// TIA Portal project "FactoryIO_Template_S7-1200_V16_V16" (V16)
// Vorlageprojekt für das Buch mit Zielsystem S7-1200

(* hardware
DEVICE "S7-1200-Station_1"  S7-1200 Station
   slot 0: "Baugruppenträger_0"  Rack  V1.0
   slot 1: "PLC_1"  CPU 1211C DC/DC/DC  6ES7 211-1AE40-0XB0  V4.1
*)

// ===== PLC "PLC_1"  CPU 1211C DC/DC/DC =====

VAR_GLOBAL   // PLC tag table "Standard-Variablentabelle"
   "6m" AT %A0.0 : Bool;
   "start" AT %E0.0 : Bool;
   "stop" AT %E0.1 : Bool;
   "Tag_4" AT %I10.0 : Bool;
   "Tag_5" AT %Q10.0 : Bool;
   "Tag_6" AT %I10.1 : Bool;
   "2m 1" AT %Q0.1 : Bool;
   "2m 2" AT %Q0.2 : Bool;
   "2m 3" AT %Q0.3 : Bool;
   "2m 4" AT %Q0.4 : Bool;
   "ccw" AT %Q0.5 : Bool;
   "sensor 4" AT %I0.3 : Bool;
   "sensor 1" AT %I0.2 : Bool;
   "pivot 1" AT %Q0.6 : Bool;
   "pivot 1 +" AT %Q0.7 : Bool;
   "sensor 2" AT %I0.4 : Bool;
   "sensor 3" AT %I0.5 : Bool;
   "pivot 2" AT %Q1.0 : Bool;
   "pivot 2 +" AT %Q1.1 : Bool;
   "pivot 3" AT %Q1.2 : Bool;
   "pivot 3 +" AT %Q1.3 : Bool;
END_VAR

// folder: System blocks/Program resources

DATA_BLOCK "IEC_Timer_0_DB"   // DB1
{ S7_Optimized_Access := 'TRUE' }
AUTHOR : Simatic
FAMILY : IEC
NAME : IEC_TMR
VERSION : 1.0
// stored: InstanceOfName IEC_TIMER
"IEC_TIMER"
BEGIN
END_DATA_BLOCK

DATA_BLOCK "IEC_Timer_0_DB_1"   // DB2
{ S7_Optimized_Access := 'TRUE' }
AUTHOR : Simatic
FAMILY : IEC
NAME : IEC_TMR
VERSION : 1.0
// stored: InstanceOfName IEC_TIMER
"IEC_TIMER"
BEGIN
END_DATA_BLOCK

DATA_BLOCK "IEC_Timer_0_DB_2"   // DB3
{ S7_Optimized_Access := 'TRUE' }
AUTHOR : Simatic
FAMILY : IEC
NAME : IEC_TMR
VERSION : 1.0
// stored: InstanceOfName IEC_TIMER
"IEC_TIMER"
BEGIN
END_DATA_BLOCK

// folder: (top level)

FUNCTION "MHJ-PLC-Lab-Function-S71200" : Void   // FC9000, SCL
{ S7_Optimized_Access := 'TRUE' }
VERSION : 0.1
   VAR_TEMP
      rdTimeReturn : Int;
      outputTime : DTL;
      SyncVal : Byte;
      forVal : Int;
      forVal_2 : Int;
      Value : Byte;
   END_VAR
   VAR CONSTANT
      CompVal : Byte := 16#34;
      Value_01 : Byte := 16#11;
      Value_01_DW : DWord := 16#A165_D992;
      Value_02_DW : DWord := 16#58BE_4401;
   END_VAR
BEGIN

   #Value:=PEEK(area := 16#82,
        dbNumber := 0,
        byteOffset := 511);
   #Value := #Value + 1;

   POKE(area := 16#82,
        dbNumber := 0,
        byteOffset := 511,
        value := #Value);

   POKE(area:=16#81,
        dbNumber:=0,
        byteOffset:=1016,
        value:=#Value_01_DW);
   POKE(area := 16#81,
        dbNumber := 0,
        byteOffset := 1020,
        value := #Value_02_DW);

   POKE(area := 16#81,
        dbNumber := 0,
        byteOffset := 511,
        value := B#16#00);

   FOR #forVal := 0 TO 120 DO
       FOR #forVal_2:=0 TO 10 DO
           #rdTimeReturn:=RD_SYS_T(#outputTime);
           #rdTimeReturn := WR_SYS_T(#outputTime);
           #rdTimeReturn := RD_SYS_T(#outputTime);
           #rdTimeReturn := WR_SYS_T(#outputTime);
       END_FOR;
       #SyncVal:= PEEK(area := 16#81,
                      dbNumber := 0,
                      byteOffset := 511);
       IF #SyncVal = #CompVal THEN
          GOTO M_1;
       END_IF;
   END_FOR;
   RETURN;

   M_1:
   POKE(area := 16#81,
        dbNumber := 0,
        byteOffset := 511,
        value := B#16#0);
END_FUNCTION

ORGANIZATION_BLOCK "Main"   // OB1, LAD, ProgramCycle
TITLE = "Main Program Sweep (Cycle)"
{ S7_Optimized_Access := 'TRUE' }
VERSION : 0.1
   VAR_INPUT
      Initial_Call : Bool;   // Initial call of this OB
      Remanence : Bool;   // =True, if remanent data are available
   END_VAR
BEGIN

REGION Network 1: Konnektierungsbaustein für PLC-Lab
   // Im Netzwerk 1 wird der Konnektierungsbaustein für PLC-Lab aufgerufen.
   // Dieser Aufruf darf nicht entfernt werden!
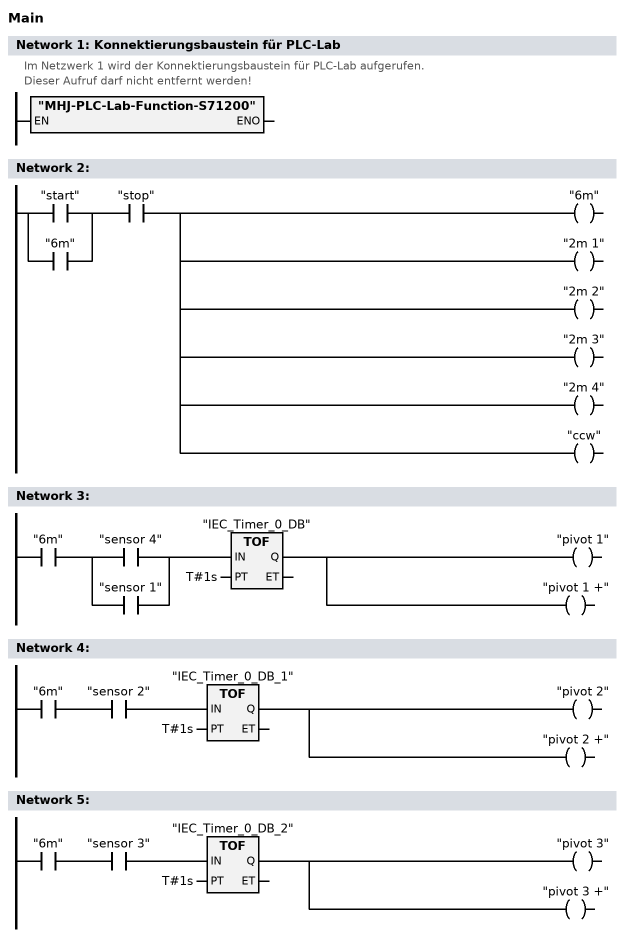
   RUNG wire#powerrail
      "MHJ-PLC-Lab-Function-S71200"()
   END_RUNG
   // the same network as SCL:
   "MHJ-PLC-Lab-Function-S71200"();
END_REGION

REGION Network 2
   RUNG wire#powerrail
      Contact( "start" )
      wire#w1
      Contact( "stop" )
      wire#w2
      Coil( "6m" )
   END_RUNG
   RUNG wire#powerrail
      Contact( "6m" )
   END_RUNG wire#w1
   RUNG wire#w2
      Coil( "2m 1" )
   END_RUNG
   RUNG wire#w2
      Coil( "2m 2" )
   END_RUNG
   RUNG wire#w2
      Coil( "2m 3" )
   END_RUNG
   RUNG wire#w2
      Coil( "2m 4" )
   END_RUNG
   RUNG wire#w2
      Coil( "ccw" )
   END_RUNG
   // the same network as SCL:
   "6m" := ("start" OR "6m") AND "stop";
   "2m 1" := "6m";
   "2m 2" := "6m";
   "2m 3" := "6m";
   "2m 4" := "6m";
   "ccw" := "6m";
END_REGION

REGION Network 3
   "IEC_Timer_0_DB".TOF(IN := "6m" AND ("sensor 4" OR "sensor 1"), PT := T#1s);
   "pivot 1" := "IEC_Timer_0_DB".Q;
   "pivot 1 +" := "IEC_Timer_0_DB".Q;
END_REGION

REGION Network 4
   "IEC_Timer_0_DB_1".TOF(IN := "6m" AND "sensor 2", PT := T#1s);
   "pivot 2" := "IEC_Timer_0_DB_1".Q;
   "pivot 2 +" := "IEC_Timer_0_DB_1".Q;
END_REGION

REGION Network 5
   "IEC_Timer_0_DB_2".TOF(IN := "6m" AND "sensor 3", PT := T#1s);
   "pivot 3" := "IEC_Timer_0_DB_2".Q;
   "pivot 3 +" := "IEC_Timer_0_DB_2".Q;
END_REGION
END_ORGANIZATION_BLOCK